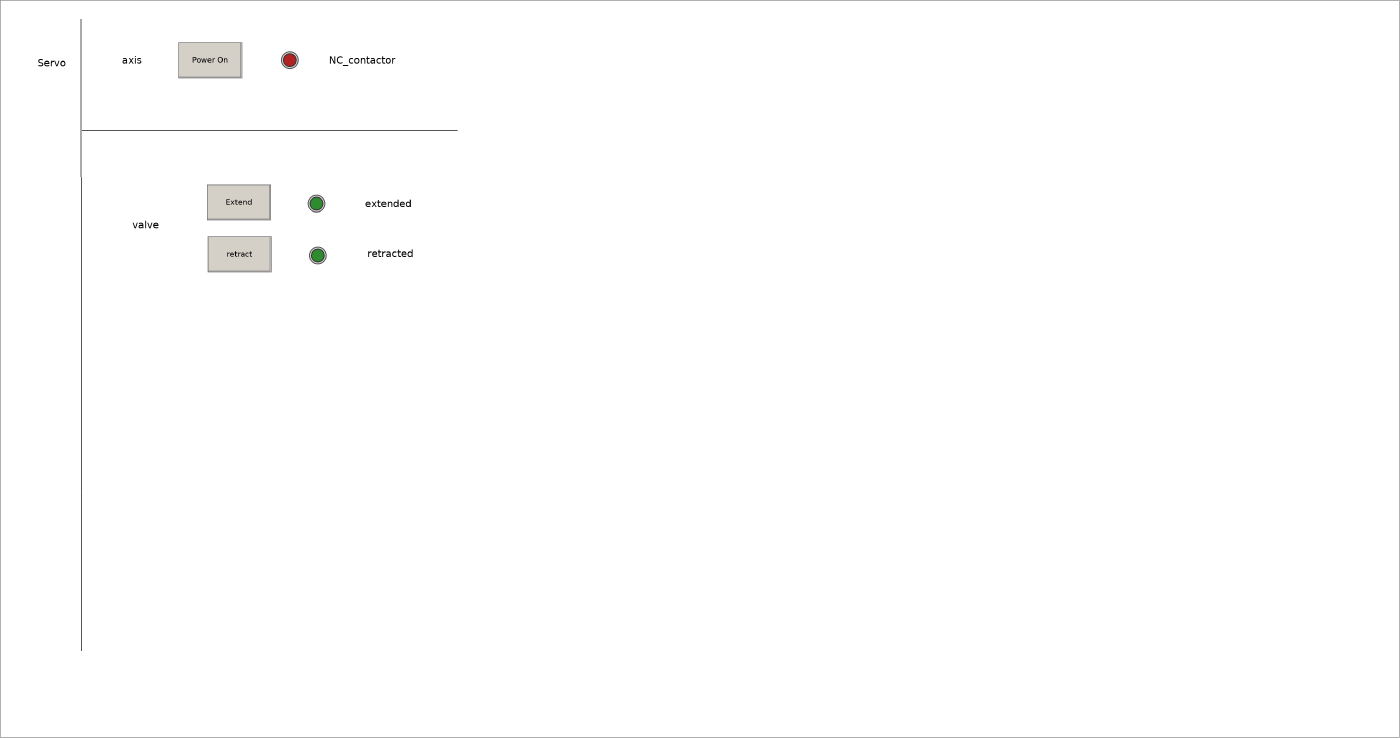
VISUALIZATION v_IO_FR  // 2048x1080
VAR_IN_OUT
	dIO_FR		: fixtureRotation_Module;
END_VAR
    Line (120,190) (669,190)
    Line (118,28) (119,952)
    Label (464,75 132x26), "NC_contactor"
    Label (127,75 132x26), "axis"
    Button (261,62 93x52), "Power On", colour toggle: dIO_FR.power_axis
        toggle dIO_FR.power_axis
    Lamp1 (409,73 30x30), variable: dIO_FR.contactor_axis, style: Lamp-Lamp1-Red
    Label (133,316 160x26), "valve"
    Button (303,270 93x52), "Extend", colour toggle: dIO_FR.valve.extend
        OnMouseDown: execute { dIO_FR.valve.extend := TRUE; dIO_FR.valve.retract := FALSE; }
    Button (304,346 93x52), "retract", colour toggle: dIO_FR.valve.retract
        OnMouseDown: execute { dIO_FR.valve.extend := FALSE; dIO_FR.valve.retract := TRUE; }
    Lamp1 (448,283 30x30), variable: dIO_FR.valve.extended, style: Lamp-Lamp1-Green
    Lamp1 (450,359 30x30), variable: dIO_FR.valve.retracted, style: Lamp-Lamp1-Green
    Label (502,285 132x26), "extended"
    Label (505,358 132x26), "retracted"
    Label (36,79 80x26), "Servo"
END_VISUALIZATION

(* stored: Version 1.1.0.1, ProductVersion 3.1.4024.12
   Visu v_IO_FR: Id {f542427b-210e-4a1e-8b88-3ce2ae3bd42d} *)
